// Block: DEBUG_MES_Receive_Msg_Topic2XX

DATA_BLOCK DEBUG_MES_Receive_Msg_Topic2XX
VERSION : 0.1
   NON_RETAIN
   VAR
      DEBUG : Struct
         Enable : Bool;
         AckChangeStep : Bool;
         ActualStep : Int;
      END_STRUCT;
      ACK_MSG_enable : Bool;
      MSG_200 : Struct
         ABILITA_FC : Bool;
         EXE_MSG : Bool;
         MSG : MES_Msg;
      END_STRUCT;
      MSG_210 : Struct
         ABILITA_FC : Bool;
         EXE_MSG : Bool;
         MSG : MES_Msg;
      END_STRUCT;
      MSG_212 : Struct
         ABILITA_FC : Bool;
         EXE_MSG : Bool;
         MSG : MES_Msg;
      END_STRUCT;
   END_VAR

BEGIN
   // No initialization required
END_DATA_BLOCK
